FUNCTION FC_ProductStatusNoPresence : eProductStatus
VAR_INPUT
	aByte					: stByteAsBit;
END_VAR

IF aByte.aBit.b1 THEN
	FC_ProductStatusNoPresence := eProductStatus.Scraped;
ELSIF aByte.aBit.b3 THEN
	FC_ProductStatusNoPresence := eProductStatus.Completed;
ELSIF aByte.aBit.b2 THEN
	FC_ProductStatusNoPresence := eProductStatus.Working;	
END_IF

END_FUNCTION

(* stored: Version 1.1.0.1, ProductVersion 3.1.4024.15
   POU FC_ProductStatusNoPresence: Id {1b1e0184-c025-40ca-b0d2-a88a20ccc013}, SpecialFunc None *)
